// TIA Portal V20 export
DATA_BLOCK "MP107"   // DB309
// stored: MemoryReserve 100
   VAR
      "MANIFOLD-1 SOL POWER MC ON" : Bool;
      "MANIFOLD-2 SOL POWER MC ON" : Bool;
      "QR LASER MARKING POWER ON 1" : Bool;
      "QR LASER MARKING POWER ON 2" : Bool;
      "FFU POWER MC ON 1" : Bool;
      "FFU POWER MC ON 2" : Bool;
      SPARE : Bool;
      SPARE_1 : Bool;
   END_VAR
BEGIN
END_DATA_BLOCK
